PROGRAM MAIN
VAR
	bQAntiBlocking:BOOL;
	bPump:BOOL;
	bError:BOOL;
	byError:BYTE;
	byState:BYTE;
	eAntiBlockingMode:E_HVACAntiBlockingMode;
	eCtrlModeActuator:E_HVACActuatorMode;
	eReqPump:E_HVACReqPump;
	sTest:STRING:='Test';
	bSetDefault:BOOL;
	bReset:BOOL;
	udiSecStopDelay:UDINT:=1;	
	udiSecFeedbPumpDelay:UDINT:=2;
	rOutsideTempHighLimit:REAL:=3.0;
	rOutsideTempLowLimit:REAL:=4.1;
	rValvePositionLimitOn:REAL:=5.2;
	rValvePositionLimitOff:REAL:=6.3;
END_VAR

IF bError THEN
	bPump := FALSE;
	byError := 2;
END_IF

IF (eCtrlModeActuator = 1 OR eCtrlModeActuator = 7) THEN
	bPump := FALSE;
END_IF

END_PROGRAM

(* stored: Version 1.1.0.1, ProductVersion 3.1.4024.3
   POU MAIN: Id {2a4304f3-537e-43d1-b89c-af5d9907262c}, SpecialFunc None *)
